// TIA Portal V19 export
DATA_BLOCK "A0303_Sollevamento"   // DB102
// stored: InstanceOfName A0303_Sollevamento_FB, InstanceOfType FB
"A0303_Sollevamento_FB"
   // VAR_INPUT
   //    AreaInterface : "AreaInterface";
   //    ZSI : "udt_ZoneSafetyInterface";
   //    DSI_Feed_Testa : "udt_DeviceSafetyInterface";
   //    DSI_Feed_Coda : "udt_DeviceSafetyInterface";
   //    DataIn : Struct
   //       OP_Vai_A_Prelievo : Bool;
   //       OP_Vai_A_Deposito : Bool;
   //       LsSensor1_Carico : Bool;
   //       LsSensor2_Carico : Bool;
   //       LsSensor1_Scarico : Bool;
   //       LsSensor2_Scarico : Bool;
   //    END_STRUCT;
   //    CIn : Struct
   //       Manager : Struct
   //          EnableStopDoorOpeningReq : Bool;
   //          EnableStopInPhase : Bool;
   //          EnableStopProgrammed : Bool;
   //          Control_ON : Bool;
   //          CanMoveFreely : Bool;
   //          TargetPosition : LReal;
   //          Phase : Struct
   //             VAI_A_PRELIEVO : Bool;
   //             VAI_A_PRE_DEPOSITO : Bool;
   //             VAI_A_DEPOSITO : Bool;
   //          END_STRUCT;
   //       END_STRUCT;
   //       Trasporto : Struct
   //          IsMeasuring : Bool;
   //       END_STRUCT;
   //    END_STRUCT;
   //    Config : Struct
   //       Testa : Struct
   //          Ax : "Positioning_DOL_Machine_Config";
   //       END_STRUCT;
   //       Coda : Struct
   //          Ax : "Positioning_DOL_Machine_Config";
   //       END_STRUCT;
   //       DelayMissingCondition { ExternalAccessible := 'False'; ExternalVisible := 'False'; ExternalWritable := 'False'} : Time;
   //    END_STRUCT;
   // END_VAR
   // VAR_OUTPUT
   //    MachineInterface : "MachineInterface";
   //    COut : Struct
   //       Ax_Testa : "Positioning_DOL_Machine_COut";
   //       Ax_Coda : "Positioning_DOL_Machine_COut";
   //       Standstill : Bool;
   //       Minus_CheckNext : Bool;
   //       Plus_CheckNext : Bool;
   //       Minus_Running : Bool;
   //       Plus_Running : Bool;
   //    END_STRUCT;
   // END_VAR
   // VAR_IN_OUT
   //    Par : Struct
   //       Ax_Man : "Positioning_DOL_Machine_Par";
   //       Ax_Testa_Pers : "Positioning_DOL_Machine_Pers_Data";
   //       Ax_Coda_Pers : "Positioning_DOL_Machine_Pers_Data";
   //       Enc : Struct
   //          Testa : "PosFbk_RTN";
   //          Coda : "PosFbk_RTN";
   //       END_STRUCT;
   //    END_STRUCT;
   //    Par_Mach : Struct
   //       PosDeposito : LReal;
   //       OffsetPrelievo : LReal;
   //       ToleranceWindow : LReal;
   //    END_STRUCT;
   // END_VAR
   // VAR
   //    Alarm : Struct
   //       Testa : Struct
   //          Ax : "Positioning_DOL_Machine_Alr";
   //          Enc { S7_SetPoint := 'True'} : "PosFbk_Encoder_Alr";
   //       END_STRUCT;
   //       Coda : Struct
   //          Ax : "Positioning_DOL_Machine_Alr";
   //          Enc { S7_SetPoint := 'True'} : "PosFbk_Encoder_Alr";
   //       END_STRUCT;
   //       CheckBothAxMove : Bool;
   //    END_STRUCT;
   //    Warning : Struct
   //       Testa : Struct
   //          Ax { S7_SetPoint := 'True'} : "Positioning_DOL_Machine_Wng";
   //       END_STRUCT;
   //       Coda : Struct
   //          Ax { S7_SetPoint := 'True'} : "Positioning_DOL_Machine_Wng";
   //       END_STRUCT;
   //       MissingCnd : Struct
   //          OP_VAI_A_PRELIEVO : Bool;
   //          OP_VAI_A_DEPOSITO : Bool;
   //       END_STRUCT;
   //    END_STRUCT;
   //    HMI : Struct
   //       Selection : Struct
   //          Ax : Int;
   //       END_STRUCT;
   //       Testa : Struct
   //          PbPreset : Bool;
   //          PresetValue : LReal;
   //       END_STRUCT;
   //       Coda : Struct
   //          PbPreset : Bool;
   //          PresetValue : LReal;
   //       END_STRUCT;
   //       PositionGraph : Int;
   //    END_STRUCT;
   //    Sts : Struct
   //       OP_CanMoveFreely : Bool;
   //       OP_Vai_A_Prelievo_Cnd : Bool;
   //       OP_Vai_A_Deposito_Cnd : Bool;
   //       OP_Vai_A_PreDeposito_Cnd : Bool;
   //       Coda_PermessoDaSynchOk : Bool;
   //       Testa_PermessoDaSynchOk : Bool;
   //    END_STRUCT;
   //    Ctrl : Struct
   //       Man : Struct
   //          OP_Vai_A_Prelievo : Bool;
   //          OP_Vai_A_Deposito : Bool;
   //       END_STRUCT;
   //       Aut : Struct
   //          OP_Vai_A_Prelievo : Bool;
   //          OP_Vai_A_Deposito : Bool;
   //          OP_Vai_A_PreDeposito : Bool;
   //       END_STRUCT;
   //       OP_Vai_A_Prelievo : Bool;
   //       OP_Vai_A_Deposito : Bool;
   //       OP_Vai_A_PreDeposito : Bool;
   //    END_STRUCT;
   //    Ax_Testa { S7_SetPoint := 'True'} : "Positioning_DOL_Machine_FB";
   //    Ax_Coda { S7_SetPoint := 'True'} : "Positioning_DOL_Machine_FB";
   //    Enc_Testa : "PosFbk_SickAFM60";
   //    Enc_Testa_ITF : "PosFbk_ITF";
   //    Enc_Coda : "PosFbk_SickAFM60";
   //    Enc_Coda_ITF : "PosFbk_ITF";
   //    AUX { ExternalAccessible := 'False'; ExternalVisible := 'False'; ExternalWritable := 'False'} : Struct
   //       OP_Vai_A_Prelievo : Bool;
   //       OP_Vai_A_Deposito : Bool;
   //    END_STRUCT;
   //    TON_OP_VAI_A_PRELIEVO_MissingCnd : IEC_TIMER;
   //    TON_OP_VAI_A_DEPOSITO_MissingCnd : IEC_TIMER;
   //    TON_CheckAxMove { S7_SetPoint := 'True'} : IEC_TIMER;
   //    TON_CheckAxis { S7_SetPoint := 'True'} : IEC_TIMER;
   //    CheckAxisSynch { S7_SetPoint := 'True'} : "CheckAxisSynch";
   //    Sts_PosAxis { S7_SetPoint := 'True'} : Int;
   // END_VAR
BEGIN
END_DATA_BLOCK
